TYPE ST_TrayProcessConfig :
STRUCT
    tLevelDetectStable : TIME; // 五层原始输入连续保持同一状态的稳定确认时间
END_STRUCT
END_TYPE

(* stored: Version 1.1.0.1, ProductVersion 3.1.4026.20
   DUT ST_TrayProcessConfig: Id {4e3ddf58-a1d2-4389-af06-07e65e71a413} *)
